// TIA Portal V19 export
TYPE "LAF_typeHmiDiagData"
TITLE = LAF_typeHmiDiagData
// HMI control tags for drive diagnostics
// stored: Access Published
   STRUCT
      referenceDesignator { ExternalWritable := 'False'} : WString[128];   // Name or reference designator of the drive object
      driveIndex : DInt;   // Selected drive object by the user during runtime in HMI
      axisStatusScreenActive : Bool;   // Axis status diagnostic screen is shown currently in HMI
      sinaStatusScreenActive : Bool;   // Sinamics status diagnostic screen is shown currently in HMI
      sinaAlarmScreenActive : Bool;   // Sinamics faults and alarm diagnostic screen is shown currently in HMI
      sinaEposScreenActive : Bool;   // Sinamics EPOS diagnostic screen is shown currently in HMI
      sinaSafetyScreenActive : Bool;   // Sinamics safety diagnostic screen is shown currently in HMI
   END_STRUCT;
END_TYPE
